TYPE EtcMasterBase_62654B43 :
STRUCT
END_STRUCT
END_TYPE

(* stored: Version 1.1.0.1, ProductVersion 3.1.4024.9
   DUT EtcMasterBase_62654B43: Id {fddc6324-06bc-4114-a736-eec440700560} *)
